INTERFACE I_Toggle EXTENDS I_RawComponent

PROPERTY IsOn : BOOL
GET
END_GET
END_PROPERTY

METHOD SwitchOff
VAR_INPUT
END_VAR
END_METHOD

METHOD SwitchOn
VAR_INPUT
END_VAR
END_METHOD

PROPERTY Tag : I_Tag
GET
END_GET
END_PROPERTY

METHOD Toggle
VAR_INPUT
END_VAR
END_METHOD

END_INTERFACE

(* stored: Version 1.1.0.1
   Itf I_Toggle: Id {1c889e8d-39df-4078-9750-0757aab29d7b}
   Property IsOn: Id {cd69bad8-da81-4d3a-969c-fe4be3ecfb6d}
   Get Get: Id {ef66c7c8-bd99-4a9d-9238-e13d8ed0cedb}
   Method SwitchOff: Id {9df1d788-b24b-45c5-bc0a-d397a005878b}
   Method SwitchOn: Id {5b9fcbe3-e2db-4f56-b465-a7b45d8fafea}
   Property Tag: Id {65706d01-ce6a-418d-884f-5549b8fbeab0}
   Get Get: Id {37bcf993-31b7-4001-8433-3cdfc8d815a4}
   Method Toggle: Id {bdb0012c-8b89-46c0-a68d-1fdf436fdbfa} *)
